REGION Network 29: High warning — Check for activation level and ON-DELAY timer
   // ▀▀▀▀▀▀▀▀▀▀▀▀▀▀▀▀▀▀▀▀▀▀▀▀▀▀▀▀▀▀▀▀▀▀▀▀▀▀▀▀▀▀▀▀
   // If the high warning has been enabled and is not masked and the actual_Value is greater than or 
   // equal to the warning setpoint (SP_WRN_H_VAL), but the warning has not yet been triggered 
   // (msg_Wrn_H = 0) then the ON-DELAY phase is active (the warning timer is counting down).
   // 
   // The timer will begin to count down from the value in TIME_WRN_H_ON_DEL using the 200ms 
   // pulse (it will count down in increments of 0.2s). If the high warning timer is less than or equal to 
   // zero, then the ON-DELAY has expired and the High warning message will become active.
   // 
   // If at any point during the ON-DELAY count down, the actual_Value drops below the activation
   // setpoint (SP_WRN_H_VAL), the timer will be reset to the TIME_WRN_H_ON_DEL value, forcing 
   // the ON-DELAY to start again.
   // ▄▄▄▄▄▄▄▄▄▄▄▄▄▄▄▄▄▄▄▄▄▄▄▄▄▄▄▄▄▄▄▄▄▄▄▄▄▄▄▄▄▄▄▄
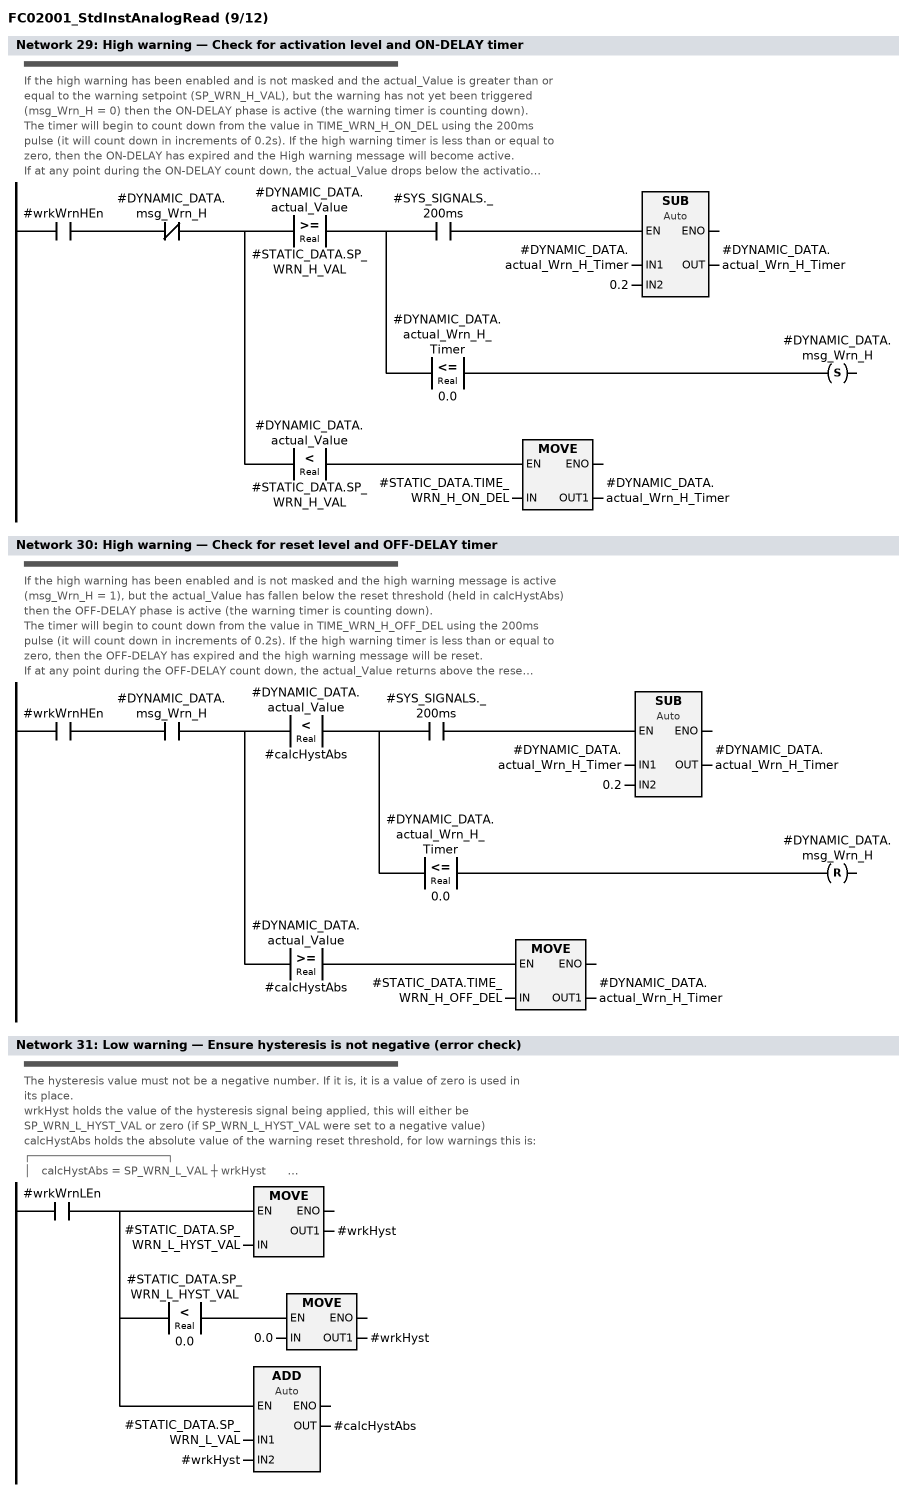
   RUNG wire#powerrail
      Contact( #wrkWrnHEn )
      I_Contact( #DYNAMIC_DATA.msg_Wrn_H )
      wire#w1
      { S7_Templates := "SrcType := Real" } GE_Contact(in1 := #DYNAMIC_DATA.actual_Value, in2 := #STATIC_DATA.SP_WRN_H_VAL)
      wire#w2
      Contact( #SYS_SIGNALS._200ms )
      Sub(in1 := #DYNAMIC_DATA.actual_Wrn_H_Timer, in2 := 0.2, out => #DYNAMIC_DATA.actual_Wrn_H_Timer)
   END_RUNG
   RUNG wire#w2
      { S7_Templates := "SrcType := Real" } LE_Contact(in1 := #DYNAMIC_DATA.actual_Wrn_H_Timer, in2 := 0.0)
      S_Coil( #DYNAMIC_DATA.msg_Wrn_H )
   END_RUNG
   RUNG wire#w1
      { S7_Templates := "SrcType := Real" } LT_Contact(in1 := #DYNAMIC_DATA.actual_Value, in2 := #STATIC_DATA.SP_WRN_H_VAL)
      { S7_GenerateENO := "TRUE" } Move(in := #STATIC_DATA.TIME_WRN_H_ON_DEL, out1 => #DYNAMIC_DATA.actual_Wrn_H_Timer)
   END_RUNG
   // the same network as SCL:
   #_w1 := #wrkWrnHEn AND NOT #DYNAMIC_DATA.msg_Wrn_H;
   #_w2 := #_w1 AND (#DYNAMIC_DATA.actual_Value >= #STATIC_DATA.SP_WRN_H_VAL);
   IF #_w2 AND #SYS_SIGNALS._200ms THEN
       #DYNAMIC_DATA.actual_Wrn_H_Timer := #DYNAMIC_DATA.actual_Wrn_H_Timer - 0.2;
   END_IF;
   IF #_w2 AND (#DYNAMIC_DATA.actual_Wrn_H_Timer <= 0.0) THEN #DYNAMIC_DATA.msg_Wrn_H := TRUE; END_IF;
   IF #_w1 AND (#DYNAMIC_DATA.actual_Value < #STATIC_DATA.SP_WRN_H_VAL) THEN
       #DYNAMIC_DATA.actual_Wrn_H_Timer := #STATIC_DATA.TIME_WRN_H_ON_DEL;
   END_IF;
END_REGION

REGION Network 30: High warning — Check for reset level and OFF-DELAY timer
   // ▀▀▀▀▀▀▀▀▀▀▀▀▀▀▀▀▀▀▀▀▀▀▀▀▀▀▀▀▀▀▀▀▀▀▀▀▀▀▀▀▀▀▀▀
   // If the high warning has been enabled and is not masked and the high warning message is active 
   // (msg_Wrn_H = 1), but the actual_Value has fallen below the reset threshold (held in calcHystAbs) 
   // then the OFF-DELAY phase is active (the warning timer is counting down).
   // 
   // The timer will begin to count down from the value in TIME_WRN_H_OFF_DEL using the 200ms 
   // pulse (it will count down in increments of 0.2s). If the high warning timer is less than or equal to 
   // zero, then the OFF-DELAY has expired and the high warning message will be reset.
   // 
   // If at any point during the OFF-DELAY count down, the actual_Value returns above the reset
   // threshold (calcHystAbs), the timer will be reset to the TIME_WRN_H_OFF_DEL value, forcing 
   // the OFF-DELAY to start again.
   // ▄▄▄▄▄▄▄▄▄▄▄▄▄▄▄▄▄▄▄▄▄▄▄▄▄▄▄▄▄▄▄▄▄▄▄▄▄▄▄▄▄▄▄▄
   RUNG wire#powerrail
      Contact( #wrkWrnHEn )
      Contact( #DYNAMIC_DATA.msg_Wrn_H )
      wire#w1
      { S7_Templates := "SrcType := Real" } LT_Contact(in1 := #DYNAMIC_DATA.actual_Value, in2 := #calcHystAbs)
      wire#w2
      Contact( #SYS_SIGNALS._200ms )
      Sub(in1 := #DYNAMIC_DATA.actual_Wrn_H_Timer, in2 := 0.2, out => #DYNAMIC_DATA.actual_Wrn_H_Timer)
   END_RUNG
   RUNG wire#w2
      { S7_Templates := "SrcType := Real" } LE_Contact(in1 := #DYNAMIC_DATA.actual_Wrn_H_Timer, in2 := 0.0)
      R_Coil( #DYNAMIC_DATA.msg_Wrn_H )
   END_RUNG
   RUNG wire#w1
      { S7_Templates := "SrcType := Real" } GE_Contact(in1 := #DYNAMIC_DATA.actual_Value, in2 := #calcHystAbs)
      { S7_GenerateENO := "TRUE" } Move(in := #STATIC_DATA.TIME_WRN_H_OFF_DEL, out1 => #DYNAMIC_DATA.actual_Wrn_H_Timer)
   END_RUNG
   // the same network as SCL:
   #_w1 := #wrkWrnHEn AND #DYNAMIC_DATA.msg_Wrn_H;
   #_w2 := #_w1 AND (#DYNAMIC_DATA.actual_Value < #calcHystAbs);
   IF #_w2 AND #SYS_SIGNALS._200ms THEN
       #DYNAMIC_DATA.actual_Wrn_H_Timer := #DYNAMIC_DATA.actual_Wrn_H_Timer - 0.2;
   END_IF;
   IF #_w2 AND (#DYNAMIC_DATA.actual_Wrn_H_Timer <= 0.0) THEN #DYNAMIC_DATA.msg_Wrn_H := FALSE; END_IF;
   IF #_w1 AND (#DYNAMIC_DATA.actual_Value >= #calcHystAbs) THEN
       #DYNAMIC_DATA.actual_Wrn_H_Timer := #STATIC_DATA.TIME_WRN_H_OFF_DEL;
   END_IF;
END_REGION

REGION Network 31: Low warning — Ensure hysteresis is not negative (error check)
   // ▀▀▀▀▀▀▀▀▀▀▀▀▀▀▀▀▀▀▀▀▀▀▀▀▀▀▀▀▀▀▀▀▀▀▀▀▀▀▀▀▀▀▀▀
   // The hysteresis value must not be a negative number. If it is, it is a value of zero is used in
   // its place.
   // 
   // wrkHyst holds the value of the hysteresis signal being applied, this will either be 
   // SP_WRN_L_HYST_VAL or zero (if SP_WRN_L_HYST_VAL were set to a negative value)
   // 
   // calcHystAbs holds the absolute value of the warning reset threshold, for low warnings this is:
   // ┌─────────────────────┐
   // │ calcHystAbs = SP_WRN_L_VAL ┼ wrkHyst    │
   // └─────────────────────┘
   // 
   // The two threshold values for the low warning are thus:
   // 
   //      Low warning activation threshold = SP_WRN_L_VAL
   //      Low warning reset threshold          = calcHystAbs
   // 
   // Note:    The hysteresis is only checked if warning is being evaluated
   // ▄▄▄▄▄▄▄▄▄▄▄▄▄▄▄▄▄▄▄▄▄▄▄▄▄▄▄▄▄▄▄▄▄▄▄▄▄▄▄▄▄▄▄▄
   RUNG wire#powerrail
      Contact( #wrkWrnLEn )
      wire#w1
      { S7_GenerateENO := "TRUE" } Move(in := #STATIC_DATA.SP_WRN_L_HYST_VAL, out1 => #wrkHyst)
   END_RUNG
   RUNG wire#w1
      { S7_Templates := "SrcType := Real" } LT_Contact(in1 := #STATIC_DATA.SP_WRN_L_HYST_VAL, in2 := 0.0)
      { S7_GenerateENO := "TRUE" } Move(in := 0.0, out1 => #wrkHyst)
   END_RUNG
   RUNG wire#w1
      Add(in1 := #STATIC_DATA.SP_WRN_L_VAL, in2 := #wrkHyst, out => #calcHystAbs)
   END_RUNG
   // the same network as SCL:
   IF #wrkWrnLEn THEN #wrkHyst := #STATIC_DATA.SP_WRN_L_HYST_VAL; END_IF;
   IF #wrkWrnLEn AND (#STATIC_DATA.SP_WRN_L_HYST_VAL < 0.0) THEN #wrkHyst := 0.0; END_IF;
   IF #wrkWrnLEn THEN #calcHystAbs := #STATIC_DATA.SP_WRN_L_VAL + #wrkHyst; END_IF;
END_REGION

REGION Network 32: Low warning — Check for activation level and ON-DELAY timer
   // ▀▀▀▀▀▀▀▀▀▀▀▀▀▀▀▀▀▀▀▀▀▀▀▀▀▀▀▀▀▀▀▀▀▀▀▀▀▀▀▀▀▀▀▀
   // If the low warning has been enabled and is not masked and the actual_Value is less than or 
   // equal to the warning setpoint (SP_WRN_L_VAL), but the warning has not yet been triggered 
   // (msg_Wrn_L = 0) then the ON-DELAY phase is active (the warning timer is counting down).
   // 
   // The timer will begin to count down from the value in TIME_WRN_L_ON_DEL using the 200ms 
   // pulse (it will count down in increments of 0.2s). If the Low warning timer is less than or equal to 
   // zero, then the ON-DELAY has expired and the Low Warning message will become active.
   // 
   // If at any point during the ON-DELAY count down, the actual_Value rises above the activation
   // setpoint (SP_WRN_L_VAL), the timer will be reset to the TIME_WRN_L_ON_DEL value, forcing 
   // the ON-DELAY to start again.
   // ▄▄▄▄▄▄▄▄▄▄▄▄▄▄▄▄▄▄▄▄▄▄▄▄▄▄▄▄▄▄▄▄▄▄▄▄▄▄▄▄▄▄▄▄
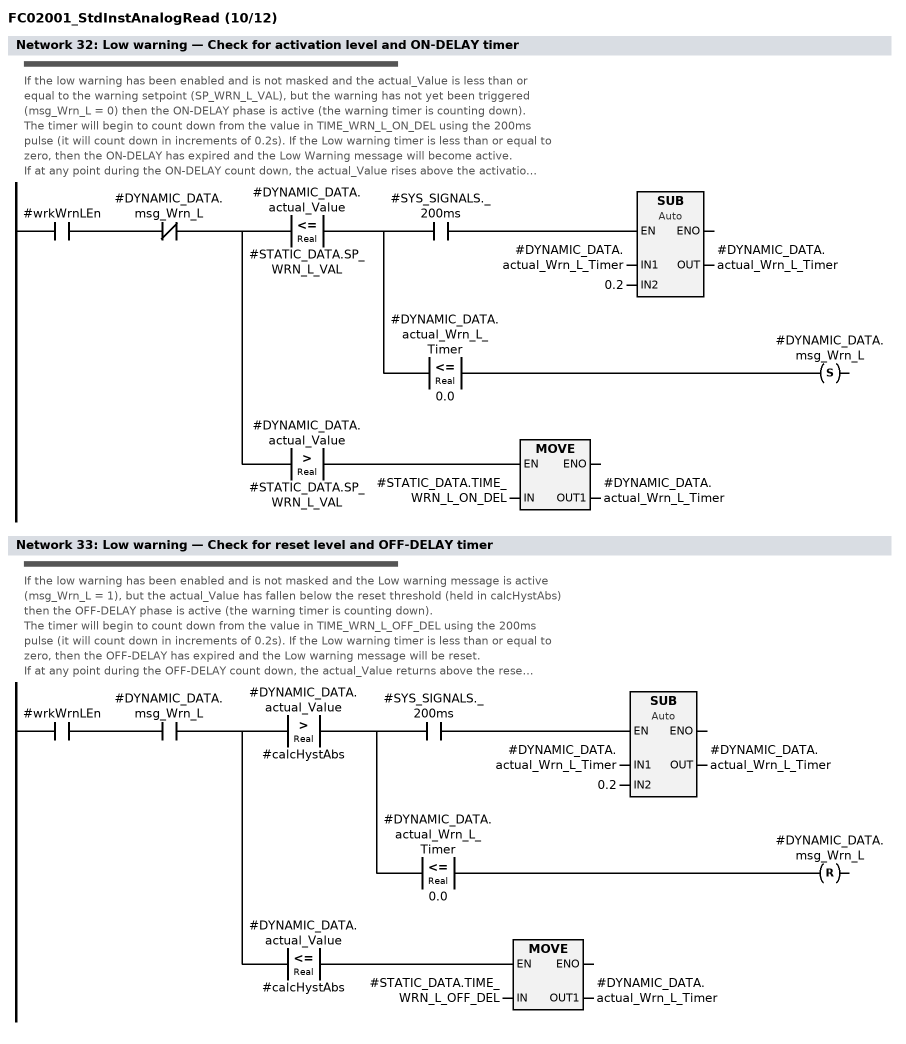
   RUNG wire#powerrail
      Contact( #wrkWrnLEn )
      I_Contact( #DYNAMIC_DATA.msg_Wrn_L )
      wire#w1
      { S7_Templates := "SrcType := Real" } LE_Contact(in1 := #DYNAMIC_DATA.actual_Value, in2 := #STATIC_DATA.SP_WRN_L_VAL)
      wire#w2
      Contact( #SYS_SIGNALS._200ms )
      Sub(in1 := #DYNAMIC_DATA.actual_Wrn_L_Timer, in2 := 0.2, out => #DYNAMIC_DATA.actual_Wrn_L_Timer)
   END_RUNG
   RUNG wire#w2
      { S7_Templates := "SrcType := Real" } LE_Contact(in1 := #DYNAMIC_DATA.actual_Wrn_L_Timer, in2 := 0.0)
      S_Coil( #DYNAMIC_DATA.msg_Wrn_L )
   END_RUNG
   RUNG wire#w1
      { S7_Templates := "SrcType := Real" } GT_Contact(in1 := #DYNAMIC_DATA.actual_Value, in2 := #STATIC_DATA.SP_WRN_L_VAL)
      { S7_GenerateENO := "TRUE" } Move(in := #STATIC_DATA.TIME_WRN_L_ON_DEL, out1 => #DYNAMIC_DATA.actual_Wrn_L_Timer)
   END_RUNG
   // the same network as SCL:
   #_w1 := #wrkWrnLEn AND NOT #DYNAMIC_DATA.msg_Wrn_L;
   #_w2 := #_w1 AND (#DYNAMIC_DATA.actual_Value <= #STATIC_DATA.SP_WRN_L_VAL);
   IF #_w2 AND #SYS_SIGNALS._200ms THEN
       #DYNAMIC_DATA.actual_Wrn_L_Timer := #DYNAMIC_DATA.actual_Wrn_L_Timer - 0.2;
   END_IF;
   IF #_w2 AND (#DYNAMIC_DATA.actual_Wrn_L_Timer <= 0.0) THEN #DYNAMIC_DATA.msg_Wrn_L := TRUE; END_IF;
   IF #_w1 AND (#DYNAMIC_DATA.actual_Value > #STATIC_DATA.SP_WRN_L_VAL) THEN
       #DYNAMIC_DATA.actual_Wrn_L_Timer := #STATIC_DATA.TIME_WRN_L_ON_DEL;
   END_IF;
END_REGION

REGION Network 33: Low warning — Check for reset level and OFF-DELAY timer
   // ▀▀▀▀▀▀▀▀▀▀▀▀▀▀▀▀▀▀▀▀▀▀▀▀▀▀▀▀▀▀▀▀▀▀▀▀▀▀▀▀▀▀▀▀
   // If the low warning has been enabled and is not masked and the Low warning message is active 
   // (msg_Wrn_L = 1), but the actual_Value has fallen below the reset threshold (held in calcHystAbs) 
   // then the OFF-DELAY phase is active (the warning timer is counting down).
   // 
   // The timer will begin to count down from the value in TIME_WRN_L_OFF_DEL using the 200ms 
   // pulse (it will count down in increments of 0.2s). If the Low warning timer is less than or equal to 
   // zero, then the OFF-DELAY has expired and the Low warning message will be reset.
   // 
   // If at any point during the OFF-DELAY count down, the actual_Value returns above the reset
   // threshold (calcHystAbs), the timer will be reset to the TIME_WRN_L_OFF_DEL value, forcing 
   // the OFF-DELAY to start again.
   // ▄▄▄▄▄▄▄▄▄▄▄▄▄▄▄▄▄▄▄▄▄▄▄▄▄▄▄▄▄▄▄▄▄▄▄▄▄▄▄▄▄▄▄▄
   RUNG wire#powerrail
      Contact( #wrkWrnLEn )
      Contact( #DYNAMIC_DATA.msg_Wrn_L )
      wire#w1
      { S7_Templates := "SrcType := Real" } GT_Contact(in1 := #DYNAMIC_DATA.actual_Value, in2 := #calcHystAbs)
      wire#w2
      Contact( #SYS_SIGNALS._200ms )
      Sub(in1 := #DYNAMIC_DATA.actual_Wrn_L_Timer, in2 := 0.2, out => #DYNAMIC_DATA.actual_Wrn_L_Timer)
   END_RUNG
   RUNG wire#w2
      { S7_Templates := "SrcType := Real" } LE_Contact(in1 := #DYNAMIC_DATA.actual_Wrn_L_Timer, in2 := 0.0)
      R_Coil( #DYNAMIC_DATA.msg_Wrn_L )
   END_RUNG
   RUNG wire#w1
      { S7_Templates := "SrcType := Real" } LE_Contact(in1 := #DYNAMIC_DATA.actual_Value, in2 := #calcHystAbs)
      { S7_GenerateENO := "TRUE" } Move(in := #STATIC_DATA.TIME_WRN_L_OFF_DEL, out1 => #DYNAMIC_DATA.actual_Wrn_L_Timer)
   END_RUNG
   // the same network as SCL:
   #_w1 := #wrkWrnLEn AND #DYNAMIC_DATA.msg_Wrn_L;
   #_w2 := #_w1 AND (#DYNAMIC_DATA.actual_Value > #calcHystAbs);
   IF #_w2 AND #SYS_SIGNALS._200ms THEN
       #DYNAMIC_DATA.actual_Wrn_L_Timer := #DYNAMIC_DATA.actual_Wrn_L_Timer - 0.2;
   END_IF;
   IF #_w2 AND (#DYNAMIC_DATA.actual_Wrn_L_Timer <= 0.0) THEN #DYNAMIC_DATA.msg_Wrn_L := FALSE; END_IF;
   IF #_w1 AND (#DYNAMIC_DATA.actual_Value <= #calcHystAbs) THEN
       #DYNAMIC_DATA.actual_Wrn_L_Timer := #STATIC_DATA.TIME_WRN_L_OFF_DEL;
   END_IF;
END_REGION

REGION Network 34: Status signals
   // ▀▀▀▀▀▀▀▀▀▀▀▀▀▀▀▀▀▀▀▀▀▀▀▀▀▀▀▀▀▀▀▀▀▀▀▀▀▀▀▀▀▀▀▀
   // The status signals for faults, alarms and warnings are either duplicates of the message signals 
   // (signals beginning with msg_) or logical combinations of them.
   // 
   // The following is a full list of the status signals:
   // 
   //  ――――――――――――――――――――――――――――――――――――――――――
   //  SIGNAL          FUNCTION            TYPE   DETAILS
   //  ――――――――――――――――――――――――――――――――――――――――――
   //  status_Alm_H       Identical to: msg_Alm_H    Bool    1 = high alm active, 0 = no alm
   // 
   //  status_Alm_L        Identical to: msg_Alm_L       Bool    1 = low alm active, 0 = no alm
   // 
   //  status_Wrn_H       Identical to: msg_Wrn_H    Bool    1 = high wrn active, 0 = no wrn
   // 
   //  status_Wrn_L        Identical to: msg_Wrn_L     Bool    1 = low wrn active, 0 = no wrn
   // 
   //  status_Alm_H_Mask     High alarm is masked        Bool    1 = alm masked, 0 = normal
   // 
   //  status_Alm_L_Mask      Low alarm is masked         Bool    1 = alm masked, 0 = normal
   // 
   //  status_Wrn_H_Mask     High warning is masked       Bool    1 = wrn masked, 0 = normal
   // 
   //  status_Wrn_L_Mask      Low warning is masked        Bool    1 = wrn masked, 0 = normal
   // 
   //  status_Alm_H_Dis         High alarm is disabled       Bool    1 = alm disabled, 0 = normal
   // 
   //  status_Alm_L_Dis          Low alarm is disabled        Bool    1 = alm disabled, 0 = normal
   // 
   //  status_Wrn_H_Dis         High warning is disabled   Bool    1 = wrn disabled, 0 = normal
   // 
   //  status_Wrn_L_Dis          Low warning is disabled       Bool    1 = wrn disabled, 0 = normal
   // 
   //  status_Fault      Indicates any of the msg_Flt    Bool    1 = fault active, 0 = healthy
   //                signals are active:
   //                  msg_Flt_UnderRange
   //                  msg_Flt_OverRange
   //                  msg_Flt_OutOfRange
   //                  msg_Flt_External 
   //                Note: msg_Flt_OutOfRange is already a combination of
   //                           msg_Flt_UnderRange and msg_Flt_OverRange
   // 
   //  status_SimOn      Status simulation mode on     Bool    1 = sim on, 0 = sim off
   // 
   //  status_RemoteOn     Status remote mode on     Bool    1 = rem on, 0 = rem off
   // 
   // 
   //  status_LocalOn      Status local mode on      Bool    1 = loc on, 0 = loc off 
   // 
   //  status_RLOff      Status ALL mode is on           Bool    1 = ALL mode on, 
   //                               0 = ALL mode off
   //  ――――――――――――――――――――――――――――――――――――――――――
   // ▄▄▄▄▄▄▄▄▄▄▄▄▄▄▄▄▄▄▄▄▄▄▄▄▄▄▄▄▄▄▄▄▄▄▄▄▄▄▄▄▄▄▄▄
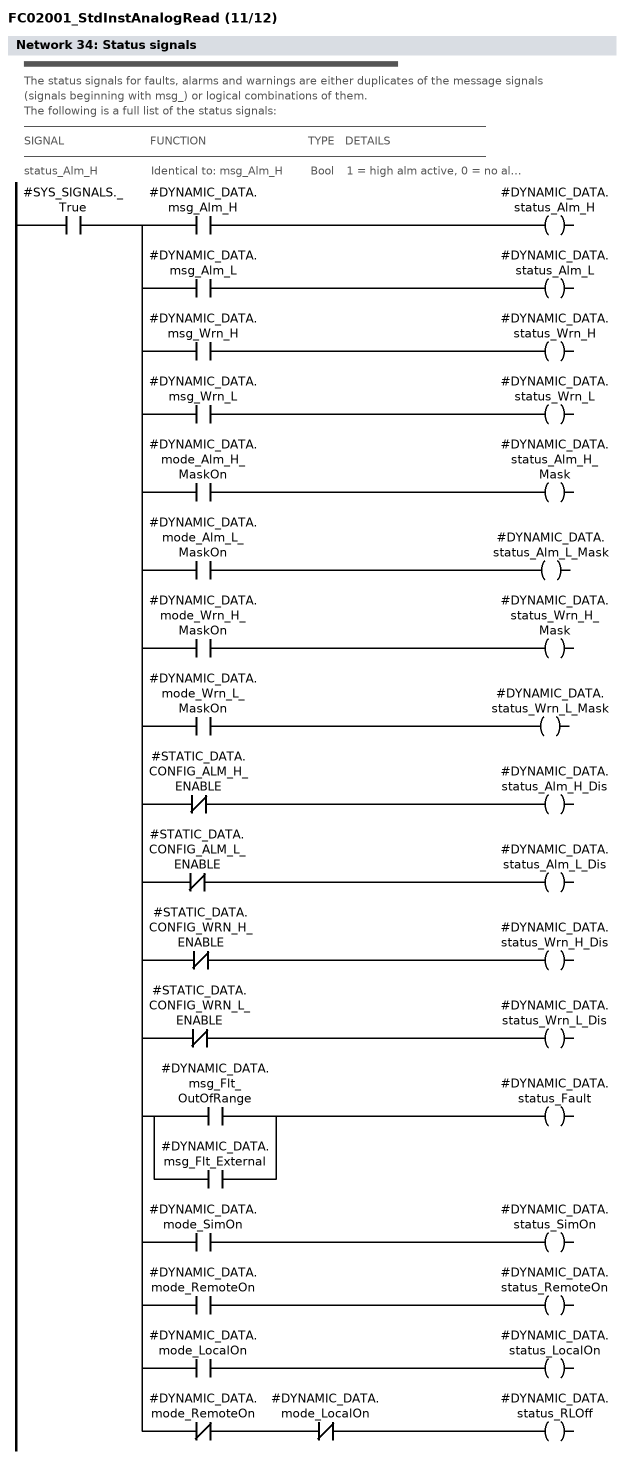
   RUNG wire#powerrail
      Contact( #SYS_SIGNALS._True )
      wire#w1
      Contact( #DYNAMIC_DATA.msg_Alm_H )
      Coil( #DYNAMIC_DATA.status_Alm_H )
   END_RUNG
   RUNG wire#w1
      Contact( #DYNAMIC_DATA.msg_Alm_L )
      Coil( #DYNAMIC_DATA.status_Alm_L )
   END_RUNG
   RUNG wire#w1
      Contact( #DYNAMIC_DATA.msg_Wrn_H )
      Coil( #DYNAMIC_DATA.status_Wrn_H )
   END_RUNG
   RUNG wire#w1
      Contact( #DYNAMIC_DATA.msg_Wrn_L )
      Coil( #DYNAMIC_DATA.status_Wrn_L )
   END_RUNG
   RUNG wire#w1
      Contact( #DYNAMIC_DATA.mode_Alm_H_MaskOn )
      Coil( #DYNAMIC_DATA.status_Alm_H_Mask )
   END_RUNG
   RUNG wire#w1
      Contact( #DYNAMIC_DATA.mode_Alm_L_MaskOn )
      Coil( #DYNAMIC_DATA.status_Alm_L_Mask )
   END_RUNG
   RUNG wire#w1
      Contact( #DYNAMIC_DATA.mode_Wrn_H_MaskOn )
      Coil( #DYNAMIC_DATA.status_Wrn_H_Mask )
   END_RUNG
   RUNG wire#w1
      Contact( #DYNAMIC_DATA.mode_Wrn_L_MaskOn )
      Coil( #DYNAMIC_DATA.status_Wrn_L_Mask )
   END_RUNG
   RUNG wire#w1
      I_Contact( #STATIC_DATA.CONFIG_ALM_H_ENABLE )
      Coil( #DYNAMIC_DATA.status_Alm_H_Dis )
   END_RUNG
   RUNG wire#w1
      I_Contact( #STATIC_DATA.CONFIG_ALM_L_ENABLE )
      Coil( #DYNAMIC_DATA.status_Alm_L_Dis )
   END_RUNG
   RUNG wire#w1
      I_Contact( #STATIC_DATA.CONFIG_WRN_H_ENABLE )
      Coil( #DYNAMIC_DATA.status_Wrn_H_Dis )
   END_RUNG
   RUNG wire#w1
      I_Contact( #STATIC_DATA.CONFIG_WRN_L_ENABLE )
      Coil( #DYNAMIC_DATA.status_Wrn_L_Dis )
   END_RUNG
   RUNG wire#w1
      Contact( #DYNAMIC_DATA.msg_Flt_OutOfRange )
      wire#w2
      Coil( #DYNAMIC_DATA.status_Fault )
   END_RUNG
   RUNG wire#w1
      Contact( #DYNAMIC_DATA.msg_Flt_External )
   END_RUNG wire#w2
   RUNG wire#w1
      Contact( #DYNAMIC_DATA.mode_SimOn )
      Coil( #DYNAMIC_DATA.status_SimOn )
   END_RUNG
   RUNG wire#w1
      Contact( #DYNAMIC_DATA.mode_RemoteOn )
      Coil( #DYNAMIC_DATA.status_RemoteOn )
   END_RUNG
   RUNG wire#w1
      Contact( #DYNAMIC_DATA.mode_LocalOn )
      Coil( #DYNAMIC_DATA.status_LocalOn )
   END_RUNG
   RUNG wire#w1
      I_Contact( #DYNAMIC_DATA.mode_RemoteOn )
      I_Contact( #DYNAMIC_DATA.mode_LocalOn )
      Coil( #DYNAMIC_DATA.status_RLOff )
   END_RUNG
   // the same network as SCL:
   #DYNAMIC_DATA.status_Alm_H := #SYS_SIGNALS._True AND #DYNAMIC_DATA.msg_Alm_H;
   #DYNAMIC_DATA.status_Alm_L := #SYS_SIGNALS._True AND #DYNAMIC_DATA.msg_Alm_L;
   #DYNAMIC_DATA.status_Wrn_H := #SYS_SIGNALS._True AND #DYNAMIC_DATA.msg_Wrn_H;
   #DYNAMIC_DATA.status_Wrn_L := #SYS_SIGNALS._True AND #DYNAMIC_DATA.msg_Wrn_L;
   #DYNAMIC_DATA.status_Alm_H_Mask := #SYS_SIGNALS._True AND #DYNAMIC_DATA.mode_Alm_H_MaskOn;
   #DYNAMIC_DATA.status_Alm_L_Mask := #SYS_SIGNALS._True AND #DYNAMIC_DATA.mode_Alm_L_MaskOn;
   #DYNAMIC_DATA.status_Wrn_H_Mask := #SYS_SIGNALS._True AND #DYNAMIC_DATA.mode_Wrn_H_MaskOn;
   #DYNAMIC_DATA.status_Wrn_L_Mask := #SYS_SIGNALS._True AND #DYNAMIC_DATA.mode_Wrn_L_MaskOn;
   #DYNAMIC_DATA.status_Alm_H_Dis := #SYS_SIGNALS._True AND NOT #STATIC_DATA.CONFIG_ALM_H_ENABLE;
   #DYNAMIC_DATA.status_Alm_L_Dis := #SYS_SIGNALS._True AND NOT #STATIC_DATA.CONFIG_ALM_L_ENABLE;
   #DYNAMIC_DATA.status_Wrn_H_Dis := #SYS_SIGNALS._True AND NOT #STATIC_DATA.CONFIG_WRN_H_ENABLE;
   #DYNAMIC_DATA.status_Wrn_L_Dis := #SYS_SIGNALS._True AND NOT #STATIC_DATA.CONFIG_WRN_L_ENABLE;
   #DYNAMIC_DATA.status_Fault := #SYS_SIGNALS._True AND (#DYNAMIC_DATA.msg_Flt_OutOfRange OR #DYNAMIC_DATA.msg_Flt_External);
   #DYNAMIC_DATA.status_SimOn := #SYS_SIGNALS._True AND #DYNAMIC_DATA.mode_SimOn;
   #DYNAMIC_DATA.status_RemoteOn := #SYS_SIGNALS._True AND #DYNAMIC_DATA.mode_RemoteOn;
   #DYNAMIC_DATA.status_LocalOn := #SYS_SIGNALS._True AND #DYNAMIC_DATA.mode_LocalOn;
   #DYNAMIC_DATA.status_RLOff := #SYS_SIGNALS._True AND NOT #DYNAMIC_DATA.mode_RemoteOn AND NOT #DYNAMIC_DATA.mode_LocalOn;
END_REGION

REGION Network 35: LICENCE AND CONTACT INFORMATION
   // ▀▀▀▀▀▀▀▀▀▀▀▀▀▀▀▀▀▀▀▀▀▀▀▀▀▀▀▀▀▀▀▀▀▀▀▀▀▀▀▀▀▀▀▀
   // LICENCE AND CONTACT INFORMATION
   // 
   // This software and its associated documentation is made available under the MIT Licence:
   // 
   // ════════════════════════════════════════════
   // 
   // The MIT License (MIT)
   // 
   // Copyright © 2020 Michael Gledhill
   // 
   // Permission is hereby granted, free of charge, to any person obtaining a copy of this software 
   // and associated documentation files (the “Software”), to deal in the Software without restriction, 
   // including without limitation the rights to use, copy, modify, merge, publish, distribute, 
   // sublicense, and/or sell copies of the Software, and to permit persons to whom the Software is 
   // furnished to do so, subject to the following conditions: 
   // 
   // The above copyright notice and this permission notice shall be included in all copies or 
   // substantial portions of the Software.
   // 
   // THE SOFTWARE IS PROVIDED “AS IS”, WITHOUT WARRANTY OF ANY KIND, EXPRESS OR IMPLIED, 
   // INCLUDING BUT NOT LIMITED TO THE WARRANTIES OF MERCHANTABILITY, FITNESS FOR A 
   // PARTICULAR PURPOSE AND NON-INFRINGEMENT. IN NO EVENT SHALL THE AUTHORS OR COPYRIGHT 
   // HOLDERS BE LIABLE FOR ANY CLAIM, DAMAGES OR OTHER LIABILITY, WHETHER IN AN ACTION OF 
   // CONTRACT, TORT OR OTHERWISE, ARISING FROM, OUT OF OR IN CONNECTION WITH THE SOFTWARE 
   // OR THE USE OR OTHER DEALINGS IN THE SOFTWARE.
   // 
   // ════════════════════════════════════════════
   //                    ┌────────────┐
   // You can reach the author by email here:   │  mg@practicalseries.com  │
   //                    └────────────┘
   // Questions, corrections, constructive criticism and complaints (polite ones) are invited.
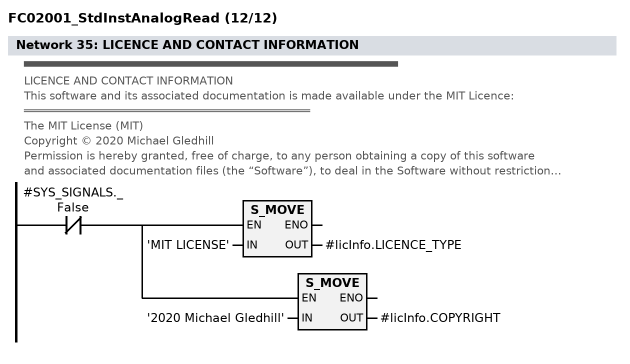
   RUNG wire#powerrail
      I_Contact( #SYS_SIGNALS._False )
      wire#w1
      S_Move(in := 'MIT LICENSE', out => #licInfo.LICENCE_TYPE)
   END_RUNG
   RUNG wire#w1
      S_Move(in := '2020 Michael Gledhill', out => #licInfo.COPYRIGHT)
   END_RUNG
   // the same network as SCL:
   IF NOT #SYS_SIGNALS._False THEN
       #licInfo.LICENCE_TYPE := 'MIT LICENSE';
       #licInfo.COPYRIGHT := '2020 Michael Gledhill';
   END_IF;
END_REGION
END_FUNCTION
